// TIA Portal V20 export
FUNCTION_BLOCK "EventsPFE"   // FB72, LAD
AUTHOR : ERsystem_FA2_DH. Kim
// stored: MemoryReserve 100, Namespace Unit1, SetENOAutomatically false
   VAR
      instResourceEvent { S7_SetPoint := 'True'} : "LPFE_ResourceEvent";
      InstTransaction1 { S7_SetPoint := 'True'} : "LER_LPFE_FNEvent";
      InstTransaction2 { S7_SetPoint := 'True'} : "LER_LPFE_FNEvent";
      InstTransaction3 { S7_SetPoint := 'True'} : "LER_LPFE_FNEvent";
      InstLPFE_ValueEvent { S7_SetPoint := 'True'} : "LPFE_ValueEvent";
      InstLPFE_TelemetryEventHandlerEM0 { S7_SetPoint := 'True'} : "LPFE_TelemetryEventHandler";
      InstLPFE_TelemetryEventHandlerEM1 { S7_SetPoint := 'True'} : "LPFE_TelemetryEventHandler";
      InstLPFE_TelemetryEventHandlerEM2 { S7_SetPoint := 'True'} : "LPFE_TelemetryEventHandler";
      InstLPFE_TelemetryEventHandlerEM3 { S7_SetPoint := 'True'} : "LPFE_TelemetryEventHandler";
      InstLPFE_TelemetryEventHandlerEM4 { S7_SetPoint := 'True'} : "LPFE_TelemetryEventHandler";
      InstLPFE_TelemetryEventHandlerEM5 { S7_SetPoint := 'True'} : "LPFE_TelemetryEventHandler";
      InstLPFE_TelemetryEventHandlerEM6 { S7_SetPoint := 'True'} : "LPFE_TelemetryEventHandler";
      InstLPFE_TelemetryEventHandlerEM7 { S7_SetPoint := 'True'} : "LPFE_TelemetryEventHandler";
      InstLPFE_RecordEvent { S7_SetPoint := 'True'} : "LPFE_RecordEvent";
   END_VAR
BEGIN

REGION Network 1: Resource Event (4)
   // Configuration example, adpat it according to the event requirements
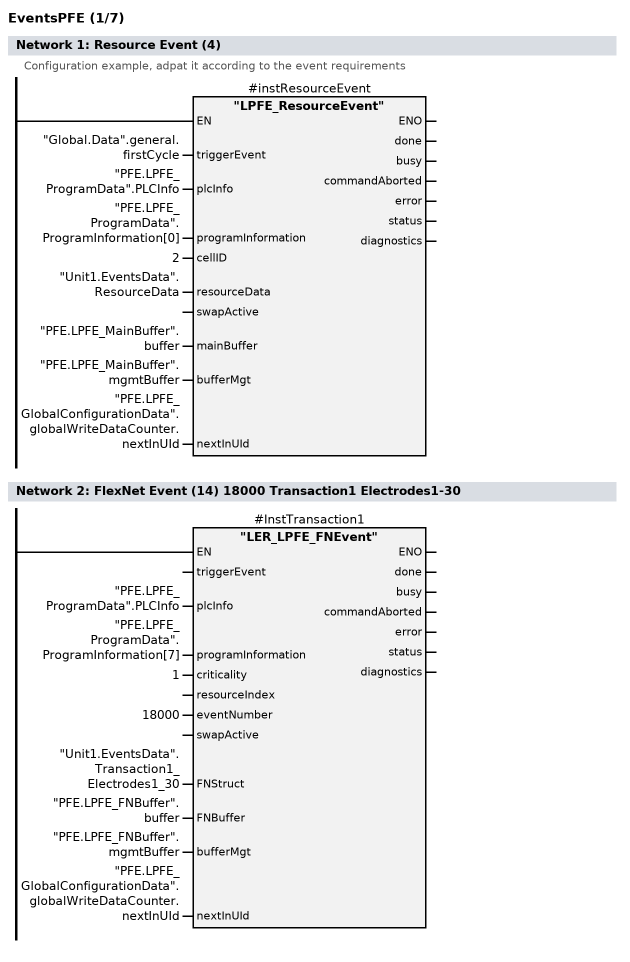
   RUNG wire#powerrail
      #instResourceEvent(triggerEvent := "Global.Data".general.firstCycle, plcInfo := "PFE.LPFE_ProgramData".PLCInfo, programInformation := "PFE.LPFE_ProgramData".ProgramInformation[0], cellID := 2, resourceData := "Unit1.EventsData".ResourceData, swapActive :=, mainBuffer := "PFE.LPFE_MainBuffer".buffer, bufferMgt := "PFE.LPFE_MainBuffer".mgmtBuffer, nextInUId := "PFE.LPFE_GlobalConfigurationData".globalWriteDataCounter.nextInUId, done =>, busy =>, commandAborted =>, error =>, status =>, diagnostics =>)
   END_RUNG
   // the same network as SCL:
   #instResourceEvent(triggerEvent := "Global.Data".general.firstCycle,   // "LPFE_ResourceEvent"
                      plcInfo := "PFE.LPFE_ProgramData".PLCInfo,
                      programInformation := "PFE.LPFE_ProgramData".ProgramInformation[0],
                      cellID := 2,
                      resourceData := "Unit1.EventsData".ResourceData,
                      mainBuffer := "PFE.LPFE_MainBuffer".buffer,
                      bufferMgt := "PFE.LPFE_MainBuffer".mgmtBuffer,
                      nextInUId := "PFE.LPFE_GlobalConfigurationData".globalWriteDataCounter.nextInUId);
END_REGION

REGION Network 2: FlexNet Event (14) 18000 Transaction1 Electrodes1-30
   RUNG wire#powerrail
      #InstTransaction1(triggerEvent :=, plcInfo := "PFE.LPFE_ProgramData".PLCInfo, programInformation := "PFE.LPFE_ProgramData".ProgramInformation[7], criticality := 1, resourceIndex :=, eventNumber := 18000, swapActive :=, FNStruct := "Unit1.EventsData".Transaction1_Electrodes1_30, FNBuffer := "PFE.LPFE_FNBuffer".buffer, bufferMgt := "PFE.LPFE_FNBuffer".mgmtBuffer, nextInUId := "PFE.LPFE_GlobalConfigurationData".globalWriteDataCounter.nextInUId, done =>, busy =>, commandAborted =>, error =>, status =>, diagnostics =>)
   END_RUNG
   // the same network as SCL:
   #InstTransaction1(plcInfo := "PFE.LPFE_ProgramData".PLCInfo,   // "LER_LPFE_FNEvent"
                     programInformation := "PFE.LPFE_ProgramData".ProgramInformation[7],
                     criticality := 1,
                     eventNumber := 18000,
                     FNStruct := "Unit1.EventsData".Transaction1_Electrodes1_30,
                     FNBuffer := "PFE.LPFE_FNBuffer".buffer,
                     bufferMgt := "PFE.LPFE_FNBuffer".mgmtBuffer,
                     nextInUId := "PFE.LPFE_GlobalConfigurationData".globalWriteDataCounter.nextInUId);
END_REGION

REGION Network 3: FlexNet Event (14) 18001 Transaction2 Electrodes31-60
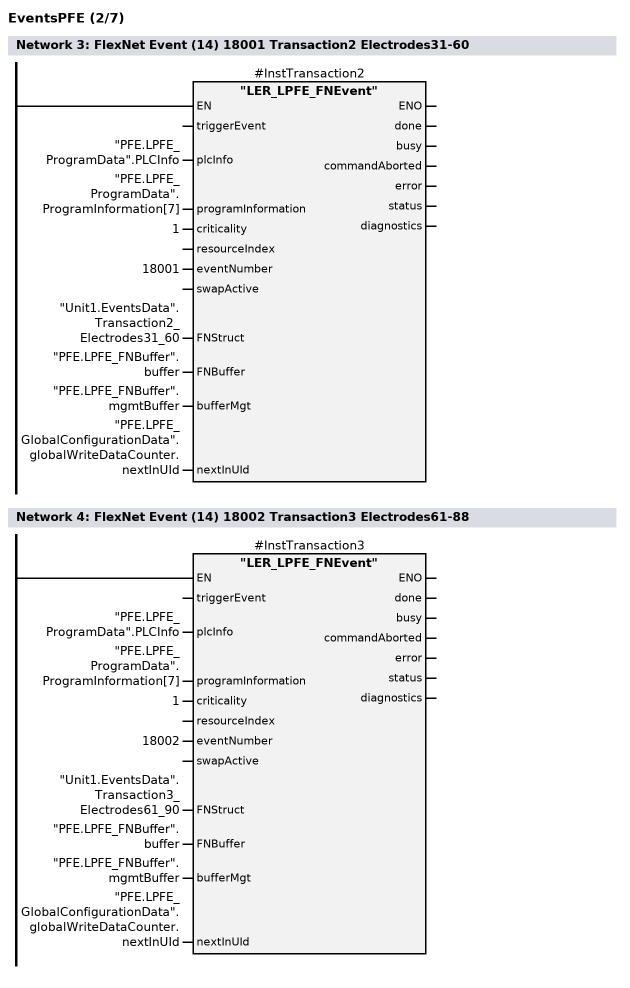
   RUNG wire#powerrail
      #InstTransaction2(triggerEvent :=, plcInfo := "PFE.LPFE_ProgramData".PLCInfo, programInformation := "PFE.LPFE_ProgramData".ProgramInformation[7], criticality := 1, resourceIndex :=, eventNumber := 18001, swapActive :=, FNStruct := "Unit1.EventsData".Transaction2_Electrodes31_60, FNBuffer := "PFE.LPFE_FNBuffer".buffer, bufferMgt := "PFE.LPFE_FNBuffer".mgmtBuffer, nextInUId := "PFE.LPFE_GlobalConfigurationData".globalWriteDataCounter.nextInUId, done =>, busy =>, commandAborted =>, error =>, status =>, diagnostics =>)
   END_RUNG
   // the same network as SCL:
   #InstTransaction2(plcInfo := "PFE.LPFE_ProgramData".PLCInfo,   // "LER_LPFE_FNEvent"
                     programInformation := "PFE.LPFE_ProgramData".ProgramInformation[7],
                     criticality := 1,
                     eventNumber := 18001,
                     FNStruct := "Unit1.EventsData".Transaction2_Electrodes31_60,
                     FNBuffer := "PFE.LPFE_FNBuffer".buffer,
                     bufferMgt := "PFE.LPFE_FNBuffer".mgmtBuffer,
                     nextInUId := "PFE.LPFE_GlobalConfigurationData".globalWriteDataCounter.nextInUId);
END_REGION

REGION Network 4: FlexNet Event (14) 18002 Transaction3 Electrodes61-88
   RUNG wire#powerrail
      #InstTransaction3(triggerEvent :=, plcInfo := "PFE.LPFE_ProgramData".PLCInfo, programInformation := "PFE.LPFE_ProgramData".ProgramInformation[7], criticality := 1, resourceIndex :=, eventNumber := 18002, swapActive :=, FNStruct := "Unit1.EventsData".Transaction3_Electrodes61_90, FNBuffer := "PFE.LPFE_FNBuffer".buffer, bufferMgt := "PFE.LPFE_FNBuffer".mgmtBuffer, nextInUId := "PFE.LPFE_GlobalConfigurationData".globalWriteDataCounter.nextInUId, done =>, busy =>, commandAborted =>, error =>, status =>, diagnostics =>)
   END_RUNG
   // the same network as SCL:
   #InstTransaction3(plcInfo := "PFE.LPFE_ProgramData".PLCInfo,   // "LER_LPFE_FNEvent"
                     programInformation := "PFE.LPFE_ProgramData".ProgramInformation[7],
                     criticality := 1,
                     eventNumber := 18002,
                     FNStruct := "Unit1.EventsData".Transaction3_Electrodes61_90,
                     FNBuffer := "PFE.LPFE_FNBuffer".buffer,
                     bufferMgt := "PFE.LPFE_FNBuffer".mgmtBuffer,
                     nextInUId := "PFE.LPFE_GlobalConfigurationData".globalWriteDataCounter.nextInUId);
END_REGION

REGION Network 5: ValueEvent (6)
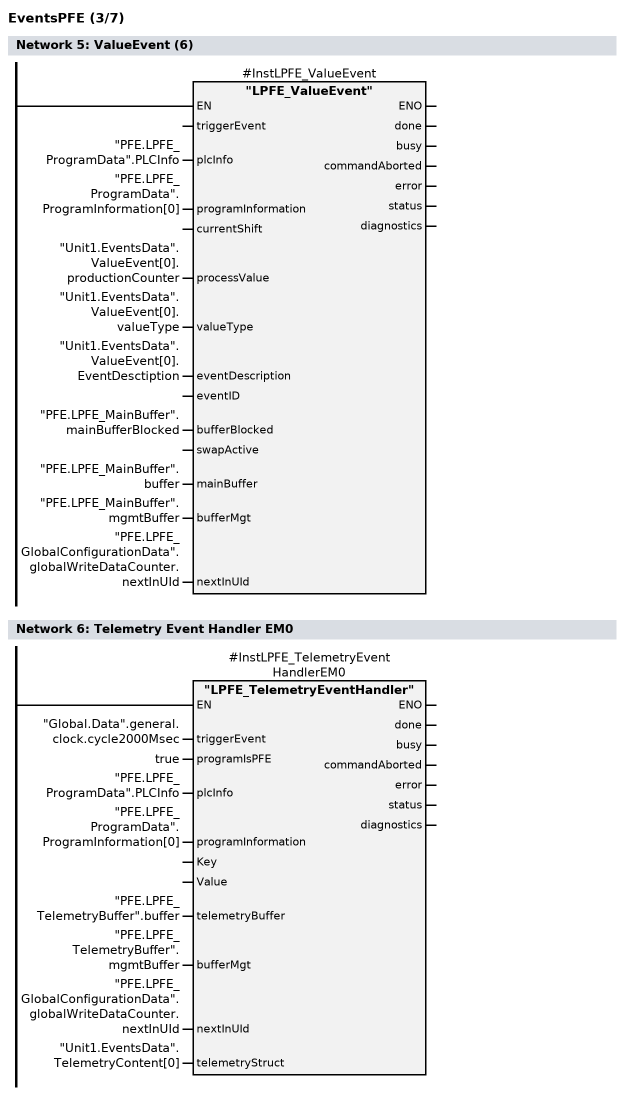
   RUNG wire#powerrail
      #InstLPFE_ValueEvent(triggerEvent :=, plcInfo := "PFE.LPFE_ProgramData".PLCInfo, programInformation := "PFE.LPFE_ProgramData".ProgramInformation[0], currentShift :=, processValue := "Unit1.EventsData".ValueEvent[0].productionCounter, valueType := "Unit1.EventsData".ValueEvent[0].valueType, eventDescription := "Unit1.EventsData".ValueEvent[0].EventDesctiption, eventID :=, bufferBlocked := "PFE.LPFE_MainBuffer".mainBufferBlocked, swapActive :=, mainBuffer := "PFE.LPFE_MainBuffer".buffer, bufferMgt := "PFE.LPFE_MainBuffer".mgmtBuffer, nextInUId := "PFE.LPFE_GlobalConfigurationData".globalWriteDataCounter.nextInUId, done =>, busy =>, commandAborted =>, error =>, status =>, diagnostics =>)
   END_RUNG
   // the same network as SCL:
   #InstLPFE_ValueEvent(plcInfo := "PFE.LPFE_ProgramData".PLCInfo,   // "LPFE_ValueEvent"
                        programInformation := "PFE.LPFE_ProgramData".ProgramInformation[0],
                        processValue := "Unit1.EventsData".ValueEvent[0].productionCounter,
                        valueType := "Unit1.EventsData".ValueEvent[0].valueType,
                        eventDescription := "Unit1.EventsData".ValueEvent[0].EventDesctiption,
                        bufferBlocked := "PFE.LPFE_MainBuffer".mainBufferBlocked,
                        mainBuffer := "PFE.LPFE_MainBuffer".buffer,
                        bufferMgt := "PFE.LPFE_MainBuffer".mgmtBuffer,
                        nextInUId := "PFE.LPFE_GlobalConfigurationData".globalWriteDataCounter.nextInUId);
END_REGION

REGION Network 6: Telemetry Event Handler EM0
   RUNG wire#powerrail
      #InstLPFE_TelemetryEventHandlerEM0(triggerEvent := "Global.Data".general.clock.cycle2000Msec, programIsPFE := true, plcInfo := "PFE.LPFE_ProgramData".PLCInfo, programInformation := "PFE.LPFE_ProgramData".ProgramInformation[0], Key :=, Value :=, telemetryBuffer := "PFE.LPFE_TelemetryBuffer".buffer, bufferMgt := "PFE.LPFE_TelemetryBuffer".mgmtBuffer, nextInUId := "PFE.LPFE_GlobalConfigurationData".globalWriteDataCounter.nextInUId, telemetryStruct := "Unit1.EventsData".TelemetryContent[0], done =>, busy =>, commandAborted =>, error =>, status =>, diagnostics =>)
   END_RUNG
   // the same network as SCL:
   #InstLPFE_TelemetryEventHandlerEM0(triggerEvent := "Global.Data".general.clock.cycle2000Msec,   // "LPFE_TelemetryEventHandler"
                           programIsPFE := true,
                           plcInfo := "PFE.LPFE_ProgramData".PLCInfo,
                           programInformation := "PFE.LPFE_ProgramData".ProgramInformation[0],
                           telemetryBuffer := "PFE.LPFE_TelemetryBuffer".buffer,
                           bufferMgt := "PFE.LPFE_TelemetryBuffer".mgmtBuffer,
                           nextInUId := "PFE.LPFE_GlobalConfigurationData".globalWriteDataCounter.nextInUId,
                           telemetryStruct := "Unit1.EventsData".TelemetryContent[0]);
END_REGION

REGION Network 7: Telemetry Event Handler EM1
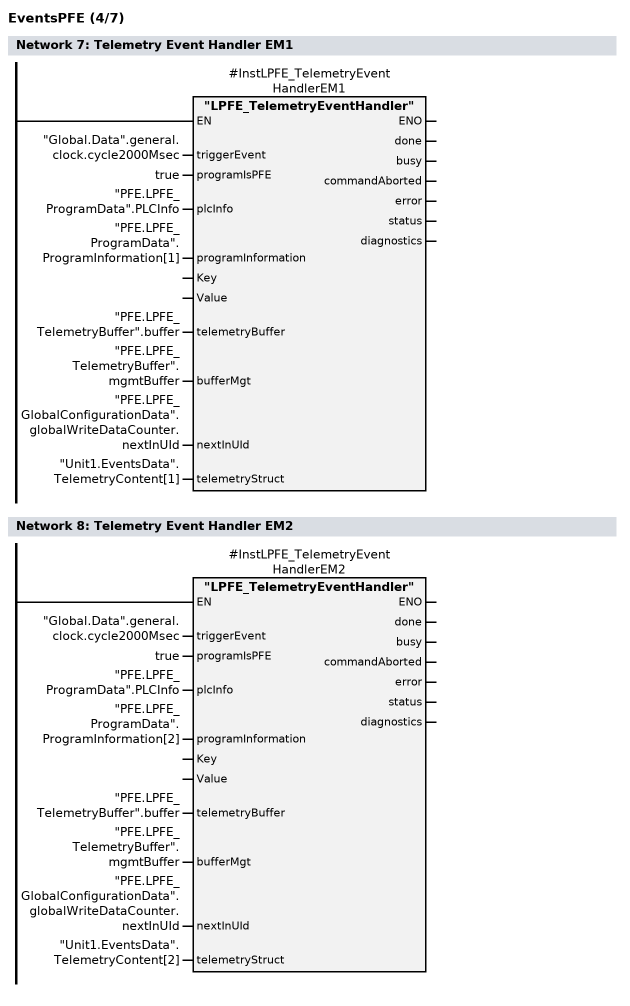
   RUNG wire#powerrail
      #InstLPFE_TelemetryEventHandlerEM1(triggerEvent := "Global.Data".general.clock.cycle2000Msec, programIsPFE := true, plcInfo := "PFE.LPFE_ProgramData".PLCInfo, programInformation := "PFE.LPFE_ProgramData".ProgramInformation[1], Key :=, Value :=, telemetryBuffer := "PFE.LPFE_TelemetryBuffer".buffer, bufferMgt := "PFE.LPFE_TelemetryBuffer".mgmtBuffer, nextInUId := "PFE.LPFE_GlobalConfigurationData".globalWriteDataCounter.nextInUId, telemetryStruct := "Unit1.EventsData".TelemetryContent[1], done =>, busy =>, commandAborted =>, error =>, status =>, diagnostics =>)
   END_RUNG
   // the same network as SCL:
   #InstLPFE_TelemetryEventHandlerEM1(triggerEvent := "Global.Data".general.clock.cycle2000Msec,   // "LPFE_TelemetryEventHandler"
                           programIsPFE := true,
                           plcInfo := "PFE.LPFE_ProgramData".PLCInfo,
                           programInformation := "PFE.LPFE_ProgramData".ProgramInformation[1],
                           telemetryBuffer := "PFE.LPFE_TelemetryBuffer".buffer,
                           bufferMgt := "PFE.LPFE_TelemetryBuffer".mgmtBuffer,
                           nextInUId := "PFE.LPFE_GlobalConfigurationData".globalWriteDataCounter.nextInUId,
                           telemetryStruct := "Unit1.EventsData".TelemetryContent[1]);
END_REGION

REGION Network 8: Telemetry Event Handler EM2
   RUNG wire#powerrail
      #InstLPFE_TelemetryEventHandlerEM2(triggerEvent := "Global.Data".general.clock.cycle2000Msec, programIsPFE := true, plcInfo := "PFE.LPFE_ProgramData".PLCInfo, programInformation := "PFE.LPFE_ProgramData".ProgramInformation[2], Key :=, Value :=, telemetryBuffer := "PFE.LPFE_TelemetryBuffer".buffer, bufferMgt := "PFE.LPFE_TelemetryBuffer".mgmtBuffer, nextInUId := "PFE.LPFE_GlobalConfigurationData".globalWriteDataCounter.nextInUId, telemetryStruct := "Unit1.EventsData".TelemetryContent[2], done =>, busy =>, commandAborted =>, error =>, status =>, diagnostics =>)
   END_RUNG
   // the same network as SCL:
   #InstLPFE_TelemetryEventHandlerEM2(triggerEvent := "Global.Data".general.clock.cycle2000Msec,   // "LPFE_TelemetryEventHandler"
                           programIsPFE := true,
                           plcInfo := "PFE.LPFE_ProgramData".PLCInfo,
                           programInformation := "PFE.LPFE_ProgramData".ProgramInformation[2],
                           telemetryBuffer := "PFE.LPFE_TelemetryBuffer".buffer,
                           bufferMgt := "PFE.LPFE_TelemetryBuffer".mgmtBuffer,
                           nextInUId := "PFE.LPFE_GlobalConfigurationData".globalWriteDataCounter.nextInUId,
                           telemetryStruct := "Unit1.EventsData".TelemetryContent[2]);
END_REGION

REGION Network 9: Telemetry Event Handler EM3
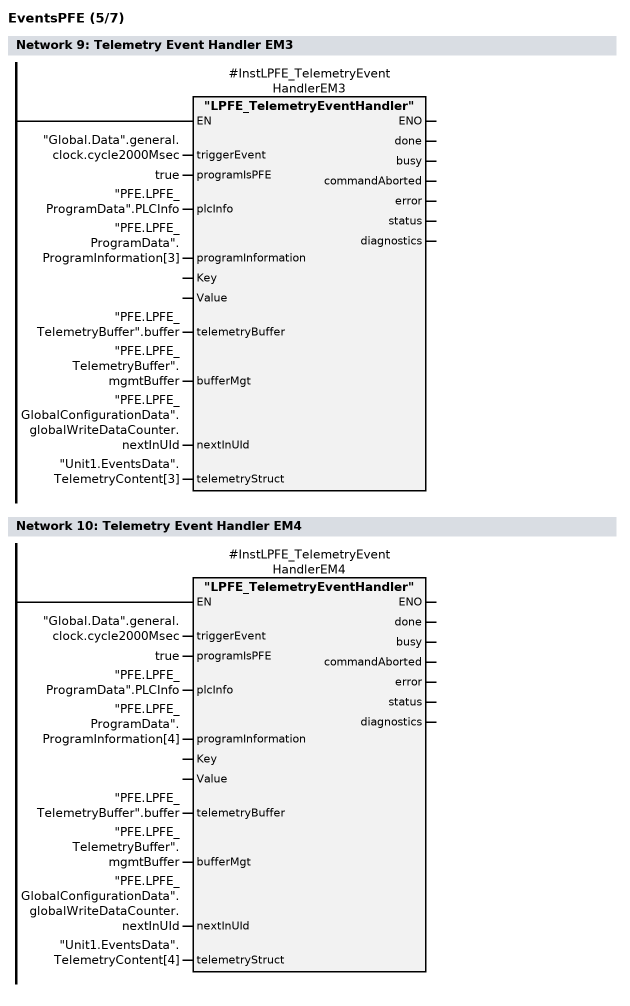
   RUNG wire#powerrail
      #InstLPFE_TelemetryEventHandlerEM3(triggerEvent := "Global.Data".general.clock.cycle2000Msec, programIsPFE := true, plcInfo := "PFE.LPFE_ProgramData".PLCInfo, programInformation := "PFE.LPFE_ProgramData".ProgramInformation[3], Key :=, Value :=, telemetryBuffer := "PFE.LPFE_TelemetryBuffer".buffer, bufferMgt := "PFE.LPFE_TelemetryBuffer".mgmtBuffer, nextInUId := "PFE.LPFE_GlobalConfigurationData".globalWriteDataCounter.nextInUId, telemetryStruct := "Unit1.EventsData".TelemetryContent[3], done =>, busy =>, commandAborted =>, error =>, status =>, diagnostics =>)
   END_RUNG
   // the same network as SCL:
   #InstLPFE_TelemetryEventHandlerEM3(triggerEvent := "Global.Data".general.clock.cycle2000Msec,   // "LPFE_TelemetryEventHandler"
                           programIsPFE := true,
                           plcInfo := "PFE.LPFE_ProgramData".PLCInfo,
                           programInformation := "PFE.LPFE_ProgramData".ProgramInformation[3],
                           telemetryBuffer := "PFE.LPFE_TelemetryBuffer".buffer,
                           bufferMgt := "PFE.LPFE_TelemetryBuffer".mgmtBuffer,
                           nextInUId := "PFE.LPFE_GlobalConfigurationData".globalWriteDataCounter.nextInUId,
                           telemetryStruct := "Unit1.EventsData".TelemetryContent[3]);
END_REGION

REGION Network 10: Telemetry Event Handler EM4
   RUNG wire#powerrail
      #InstLPFE_TelemetryEventHandlerEM4(triggerEvent := "Global.Data".general.clock.cycle2000Msec, programIsPFE := true, plcInfo := "PFE.LPFE_ProgramData".PLCInfo, programInformation := "PFE.LPFE_ProgramData".ProgramInformation[4], Key :=, Value :=, telemetryBuffer := "PFE.LPFE_TelemetryBuffer".buffer, bufferMgt := "PFE.LPFE_TelemetryBuffer".mgmtBuffer, nextInUId := "PFE.LPFE_GlobalConfigurationData".globalWriteDataCounter.nextInUId, telemetryStruct := "Unit1.EventsData".TelemetryContent[4], done =>, busy =>, commandAborted =>, error =>, status =>, diagnostics =>)
   END_RUNG
   // the same network as SCL:
   #InstLPFE_TelemetryEventHandlerEM4(triggerEvent := "Global.Data".general.clock.cycle2000Msec,   // "LPFE_TelemetryEventHandler"
                           programIsPFE := true,
                           plcInfo := "PFE.LPFE_ProgramData".PLCInfo,
                           programInformation := "PFE.LPFE_ProgramData".ProgramInformation[4],
                           telemetryBuffer := "PFE.LPFE_TelemetryBuffer".buffer,
                           bufferMgt := "PFE.LPFE_TelemetryBuffer".mgmtBuffer,
                           nextInUId := "PFE.LPFE_GlobalConfigurationData".globalWriteDataCounter.nextInUId,
                           telemetryStruct := "Unit1.EventsData".TelemetryContent[4]);
END_REGION

REGION Network 11: Telemetry Event Handler EM5
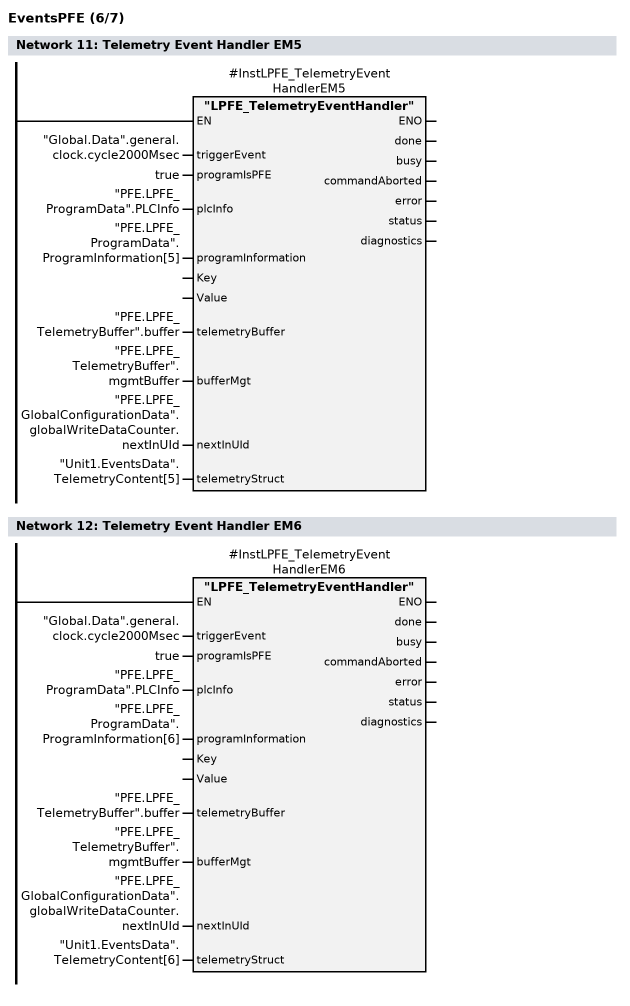
   RUNG wire#powerrail
      #InstLPFE_TelemetryEventHandlerEM5(triggerEvent := "Global.Data".general.clock.cycle2000Msec, programIsPFE := true, plcInfo := "PFE.LPFE_ProgramData".PLCInfo, programInformation := "PFE.LPFE_ProgramData".ProgramInformation[5], Key :=, Value :=, telemetryBuffer := "PFE.LPFE_TelemetryBuffer".buffer, bufferMgt := "PFE.LPFE_TelemetryBuffer".mgmtBuffer, nextInUId := "PFE.LPFE_GlobalConfigurationData".globalWriteDataCounter.nextInUId, telemetryStruct := "Unit1.EventsData".TelemetryContent[5], done =>, busy =>, commandAborted =>, error =>, status =>, diagnostics =>)
   END_RUNG
   // the same network as SCL:
   #InstLPFE_TelemetryEventHandlerEM5(triggerEvent := "Global.Data".general.clock.cycle2000Msec,   // "LPFE_TelemetryEventHandler"
                           programIsPFE := true,
                           plcInfo := "PFE.LPFE_ProgramData".PLCInfo,
                           programInformation := "PFE.LPFE_ProgramData".ProgramInformation[5],
                           telemetryBuffer := "PFE.LPFE_TelemetryBuffer".buffer,
                           bufferMgt := "PFE.LPFE_TelemetryBuffer".mgmtBuffer,
                           nextInUId := "PFE.LPFE_GlobalConfigurationData".globalWriteDataCounter.nextInUId,
                           telemetryStruct := "Unit1.EventsData".TelemetryContent[5]);
END_REGION

REGION Network 12: Telemetry Event Handler EM6
   RUNG wire#powerrail
      #InstLPFE_TelemetryEventHandlerEM6(triggerEvent := "Global.Data".general.clock.cycle2000Msec, programIsPFE := true, plcInfo := "PFE.LPFE_ProgramData".PLCInfo, programInformation := "PFE.LPFE_ProgramData".ProgramInformation[6], Key :=, Value :=, telemetryBuffer := "PFE.LPFE_TelemetryBuffer".buffer, bufferMgt := "PFE.LPFE_TelemetryBuffer".mgmtBuffer, nextInUId := "PFE.LPFE_GlobalConfigurationData".globalWriteDataCounter.nextInUId, telemetryStruct := "Unit1.EventsData".TelemetryContent[6], done =>, busy =>, commandAborted =>, error =>, status =>, diagnostics =>)
   END_RUNG
   // the same network as SCL:
   #InstLPFE_TelemetryEventHandlerEM6(triggerEvent := "Global.Data".general.clock.cycle2000Msec,   // "LPFE_TelemetryEventHandler"
                           programIsPFE := true,
                           plcInfo := "PFE.LPFE_ProgramData".PLCInfo,
                           programInformation := "PFE.LPFE_ProgramData".ProgramInformation[6],
                           telemetryBuffer := "PFE.LPFE_TelemetryBuffer".buffer,
                           bufferMgt := "PFE.LPFE_TelemetryBuffer".mgmtBuffer,
                           nextInUId := "PFE.LPFE_GlobalConfigurationData".globalWriteDataCounter.nextInUId,
                           telemetryStruct := "Unit1.EventsData".TelemetryContent[6]);
END_REGION

REGION Network 13: Telemetry Event Handler EM7
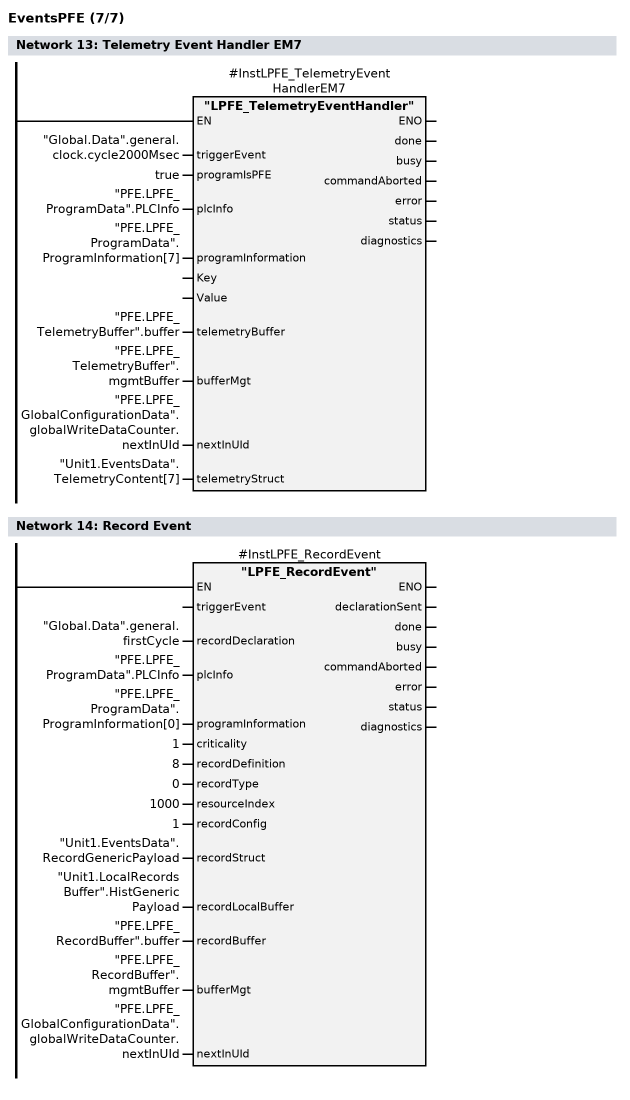
   RUNG wire#powerrail
      #InstLPFE_TelemetryEventHandlerEM7(triggerEvent := "Global.Data".general.clock.cycle2000Msec, programIsPFE := true, plcInfo := "PFE.LPFE_ProgramData".PLCInfo, programInformation := "PFE.LPFE_ProgramData".ProgramInformation[7], Key :=, Value :=, telemetryBuffer := "PFE.LPFE_TelemetryBuffer".buffer, bufferMgt := "PFE.LPFE_TelemetryBuffer".mgmtBuffer, nextInUId := "PFE.LPFE_GlobalConfigurationData".globalWriteDataCounter.nextInUId, telemetryStruct := "Unit1.EventsData".TelemetryContent[7], done =>, busy =>, commandAborted =>, error =>, status =>, diagnostics =>)
   END_RUNG
   // the same network as SCL:
   #InstLPFE_TelemetryEventHandlerEM7(triggerEvent := "Global.Data".general.clock.cycle2000Msec,   // "LPFE_TelemetryEventHandler"
                           programIsPFE := true,
                           plcInfo := "PFE.LPFE_ProgramData".PLCInfo,
                           programInformation := "PFE.LPFE_ProgramData".ProgramInformation[7],
                           telemetryBuffer := "PFE.LPFE_TelemetryBuffer".buffer,
                           bufferMgt := "PFE.LPFE_TelemetryBuffer".mgmtBuffer,
                           nextInUId := "PFE.LPFE_GlobalConfigurationData".globalWriteDataCounter.nextInUId,
                           telemetryStruct := "Unit1.EventsData".TelemetryContent[7]);
END_REGION

REGION Network 14: Record Event
   RUNG wire#powerrail
      #InstLPFE_RecordEvent(triggerEvent :=, recordDeclaration := "Global.Data".general.firstCycle, plcInfo := "PFE.LPFE_ProgramData".PLCInfo, programInformation := "PFE.LPFE_ProgramData".ProgramInformation[0], criticality := 1, recordDefinition := 8, recordType := 0, resourceIndex := 1000, recordConfig := 1, recordStruct := "Unit1.EventsData".RecordGenericPayload, recordLocalBuffer := "Unit1.LocalRecordsBuffer".HistGenericPayload, recordBuffer := "PFE.LPFE_RecordBuffer".buffer, bufferMgt := "PFE.LPFE_RecordBuffer".mgmtBuffer, nextInUId := "PFE.LPFE_GlobalConfigurationData".globalWriteDataCounter.nextInUId, declarationSent =>, done =>, busy =>, commandAborted =>, error =>, status =>, diagnostics =>)
   END_RUNG
   // the same network as SCL:
   #InstLPFE_RecordEvent(recordDeclaration := "Global.Data".general.firstCycle,   // "LPFE_RecordEvent"
                         plcInfo := "PFE.LPFE_ProgramData".PLCInfo,
                         programInformation := "PFE.LPFE_ProgramData".ProgramInformation[0],
                         criticality := 1,
                         recordDefinition := 8,
                         recordType := 0,
                         resourceIndex := 1000,
                         recordConfig := 1,
                         recordStruct := "Unit1.EventsData".RecordGenericPayload,
                         recordLocalBuffer := "Unit1.LocalRecordsBuffer".HistGenericPayload,
                         recordBuffer := "PFE.LPFE_RecordBuffer".buffer,
                         bufferMgt := "PFE.LPFE_RecordBuffer".mgmtBuffer,
                         nextInUId := "PFE.LPFE_GlobalConfigurationData".globalWriteDataCounter.nextInUId);
END_REGION

REGION Network 15: End of the Structure
END_REGION
END_FUNCTION_BLOCK
